{attribute 'qualified_only'}
VAR_GLOBAL
	bReset 		AT%Q*	:BOOL;
	bSON 		AT%Q*	:BOOL;
	bCW 		AT%Q*	:BOOL;
	bCCW 		AT%Q*	:BOOL;
	iInVoltage  AT%Q*	:INT;
END_VAR

(* stored: Version 1.1.0.1, ProductVersion 3.1.4026.6
   GVL MR_J_Motor: Id {b85c43ea-4ba9-441c-b68d-302d9ff92c66} *)
